// TIA Portal V17 export
// export: Created 2022-07-20T07:01:26.6168185Z, ExportSetting WithDefaults, DisplayName Totally Integrated Automation Portal, DisplayVersion V17, DisplayName TIA Portal Openness, DisplayVersion V17, DisplayName TIA Portal Version Control Interface, DisplayVersion V17, DisplayName SINAMICS Startdrive Advanced, DisplayVersion V17, DisplayName SINAMICS Startdrive G130, G150, S120, S150, SINAMICS MV, S210, DisplayVersion V17, DisplayName SINAMICS Startdrive G110M, G120, G120C, G120D, G120P, G115D, DisplayVersion V17, DisplayName STEP 7 Professional, DisplayVersion V17, DisplayName STEP 7 Safety, DisplayVersion V17, DisplayName WinCC Advanced, DisplayVersion V17
FUNCTION_BLOCK "FB10234_LexiumMotor"   // FB10234, LAD
{ S7_Optimized_Access := 'TRUE' }
VERSION : 0.1
// stored: AutoNumber false, IsIECCheckEnabled false, IsRetainMemResEnabled false, MemoryReserve 100, SetENOAutomatically false, UDAEnableTagReadback false
   VAR_INPUT
      Drive_In : "TLexium_MDrv_Drv2Plc";
      RequestAcknowledge : Bool;
      RequestHoming : Bool;
      ScaleInverted : Bool;
      RequestGoToAbsolutePosition_1 : Bool;
      RequestGoToAbsolutePosition_2 : Bool;
      RequestGoToAbsolutePosition_3 : Bool;
      RequestGoToAbsolutePosition_4 : Bool;
      RequestGoToAbsolutePosition_5 : Bool;
      RequestGoToAbsolutePosition_6 : Bool;
      RequestGoToAbsolutePosition_7 : Bool;
      RequestGoToAbsolutePosition_8 : Bool;
      RequestGoToAbsolutePosition_9 : Bool;
      RequestGoToAbsolutePosition_10 : Bool;
      RequestGoToRelativePosition : Bool;
      RequestJogBackward : Bool;
      RequestJogForward : Bool;
      RequestStop : Bool;
      AbsolutePosition_1 : Real;
      AbsolutePosition_2 : Real;
      AbsolutePosition_3 : Real;
      AbsolutePosition_4 : Real;
      AbsolutePosition_5 : Real;
      AbsolutePosition_6 : Real;
      AbsolutePosition_7 : Real;
      AbsolutePosition_8 : Real;
      AbsolutePosition_9 : Real;
      AbsolutePosition_10 : Real;
      HoldCurrent : SInt;
      RunCurrent : SInt;
      StepResolution : UInt := 25;
      StepsByMotorTurn : DInt := 200;
      MmByMotorTurn : LReal;
      "InitialVelocity_mm.s-1" : Real;
      "HomingVelocity_mm.s-1" : DInt;
      "Velocity_mm.s-1" : Real;
      "JogVelocity_mm.s-1" : Real;
      "Acceleration_mm.s-2" : Real;
      "Deceleration_mm.s-2" : Real;
   END_VAR
   VAR_OUTPUT
      ActualPosition_mm : Real;
      MotorInMovement : Bool;
      HomingInProgress : Bool;
      HomingDone : Bool;
      IsInAbsolutePosition_1 { ExternalAccessible := 'False'; ExternalVisible := 'False'; ExternalWritable := 'False'} : Bool;
      IsInAbsolutePosition_2 { ExternalAccessible := 'False'; ExternalVisible := 'False'; ExternalWritable := 'False'} : Bool;
      IsInAbsolutePosition_3 { ExternalAccessible := 'False'; ExternalVisible := 'False'; ExternalWritable := 'False'} : Bool;
      IsInAbsolutePosition_4 { ExternalAccessible := 'False'; ExternalVisible := 'False'; ExternalWritable := 'False'} : Bool;
      IsInAbsolutePosition_5 { ExternalAccessible := 'False'; ExternalVisible := 'False'; ExternalWritable := 'False'} : Bool;
      IsInAbsolutePosition_6 { ExternalAccessible := 'False'; ExternalVisible := 'False'; ExternalWritable := 'False'} : Bool;
      IsInAbsolutePosition_7 { ExternalAccessible := 'False'; ExternalVisible := 'False'; ExternalWritable := 'False'} : Bool;
      IsInAbsolutePosition_8 { ExternalAccessible := 'False'; ExternalVisible := 'False'; ExternalWritable := 'False'} : Bool;
      IsInAbsolutePosition_9 { ExternalAccessible := 'False'; ExternalVisible := 'False'; ExternalWritable := 'False'} : Bool;
      IsInAbsolutePosition_10 { ExternalAccessible := 'False'; ExternalVisible := 'False'; ExternalWritable := 'False'} : Bool;
      IsInAbsoluteMicrostepPosition_1 : Bool;
      IsInAbsoluteMicrostepPosition_2 : Bool;
      IsInAbsoluteMicrostepPosition_3 : Bool;
      IsInAbsoluteMicrostepPosition_4 : Bool;
      IsInAbsoluteMicrostepPosition_5 : Bool;
      IsInAbsoluteMicrostepPosition_6 : Bool;
      IsInAbsoluteMicrostepPosition_7 : Bool;
      IsInAbsoluteMicrostepPosition_8 : Bool;
      IsInAbsoluteMicrostepPosition_9 : Bool;
      IsInAbsoluteMicrostepPosition_10 : Bool;
      Busy : Bool;
      StatusCode : UInt;
      Error : Bool;
      ErrorCode : Array[0..9] of UInt;
   END_VAR
   VAR_IN_OUT
      Drive_Out : "TLexium_MDrv_Plc2Drv";
   END_VAR
   VAR
      SendJog : Bool;
      Static_InError : Bool;
      HomingErrorDetected : Bool;
      AcknowledgeHomingError : Bool;
      AcknowledgeStopError : Bool;
      SendHomingType : Bool;
      SendHomingPosition : Bool;
      SendAbsolutePosition : Bool;
      LockedRotorFaultDetected : Bool;
      i : USInt;
      NumberOfErrorDetected : USInt;
      MotorMovementStateDiagram : Int;
      Static_ErrorCode : UInt;
      MaxVelocity : DWord;
      AbsoluteMicrostepPosition_1 : LInt;
      AbsoluteMicrostepPosition_2 : LInt;
      AbsoluteMicrostepPosition_3 : LInt;
      AbsoluteMicrostepPosition_4 : LInt;
      AbsoluteMicrostepPosition_5 : LInt;
      AbsoluteMicrostepPosition_6 : LInt;
      AbsoluteMicrostepPosition_7 : LInt;
      AbsoluteMicrostepPosition_8 : LInt;
      AbsoluteMicrostepPosition_9 : LInt;
      AbsoluteMicrostepPosition_10 : LInt;
      R_TRIG_MotorAcknowledge : R_TRIG;
      R_TRIG_ChangeMicrostepResolution : R_TRIG;
      R_TRIG_ChangeInitialVelocity : R_TRIG;
      R_TRIG_ChangeVelocity : R_TRIG;
      R_TRIG_ChangeJogVelocity : R_TRIG;
      R_TRIG_ChangeAcceleration : R_TRIG;
      R_TRIG_ChangeDeceleration { S7_SetPoint := 'True'} : R_TRIG;
      R_TRIG_ChangeRunCurrent : R_TRIG;
      R_TRIG_ChangeHoldCurrent : R_TRIG;
      R_TRIG_RequestHoming { S7_SetPoint := 'True'} : R_TRIG;
      R_TRIG_RequestGoToPosition_1 { S7_SetPoint := 'True'} : R_TRIG;
      R_TRIG_RequestGoToPosition_2 { S7_SetPoint := 'True'} : R_TRIG;
      R_TRIG_RequestGoToPosition_3 { S7_SetPoint := 'True'} : R_TRIG;
      R_TRIG_RequestGoToPosition_4 { S7_SetPoint := 'True'} : R_TRIG;
      R_TRIG_RequestGoToPosition_5 { S7_SetPoint := 'True'} : R_TRIG;
      R_TRIG_RequestGoToPosition_6 { S7_SetPoint := 'True'} : R_TRIG;
      R_TRIG_RequestGoToPosition_7 { S7_SetPoint := 'True'} : R_TRIG;
      R_TRIG_RequestGoToPosition_8 { S7_SetPoint := 'True'} : R_TRIG;
      R_TRIG_RequestGoToPosition_9 { S7_SetPoint := 'True'} : R_TRIG;
      R_TRIG_RequestGoToPosition_10 { S7_SetPoint := 'True'} : R_TRIG;
      R_TRIG_RequestJogForward { S7_SetPoint := 'True'} : R_TRIG;
      R_TRIG_RequestJogBackward { S7_SetPoint := 'True'} : R_TRIG;
      R_TRIG_RequestStop { S7_SetPoint := 'True'} : R_TRIG;
      R_TRIG_MotorStopped { S7_SetPoint := 'True'} : R_TRIG;
      R_TRIG_MotorMovementDone { S7_SetPoint := 'True'} : R_TRIG;
      R_TRIG_ScaleInverted { S7_SetPoint := 'True'} : R_TRIG;
      R_TRIG_ErrorCodeChanged { S7_SetPoint := 'True'} : R_TRIG;
      R_TRIG_HomingErrorDetected { S7_SetPoint := 'True'} : R_TRIG;
      F_TRIG_RequestJogForward { S7_SetPoint := 'True'} : F_TRIG;
      F_TRIG_RequestJogBackward { S7_SetPoint := 'True'} : F_TRIG;
      TON_MotorHM { S7_SetPoint := 'True'} : TON_TIME;
      TON_MotorEnabled : TON_TIME;
      TON_MotorNotEnabled { S7_SetPoint := 'True'} : TOF_TIME;
      TON_MotorNotMoving { S7_SetPoint := 'True'} : TOF_TIME;
      TON_MotorHomingMovementDone { S7_SetPoint := 'True'} : TON_TIME;
      TON_MotorStopped { S7_SetPoint := 'True'} : TON_TIME;
      TON_IsInAbsolutePosition { S7_SetPoint := 'True'} : TON_TIME;
      TON_RetractSensorTimeout { S7_SetPoint := 'True'} : TON_TIME;
      FB10003_Pulse_SendHoldCurrent { S7_SetPoint := 'True'} : "FB10003_Pulse";
      FB10003_Pulse_SendRunCurrent { S7_SetPoint := 'True'} : "FB10003_Pulse";
      FB10003_Pulse_SendDeceleration { S7_SetPoint := 'True'} : "FB10003_Pulse";
      FB10003_Pulse_SendAcceleration { S7_SetPoint := 'True'} : "FB10003_Pulse";
      FB10003_Pulse_SendMicrostepResolution { S7_SetPoint := 'True'} : "FB10003_Pulse";
      FB10003_Pulse_SendInitialVelocity { S7_SetPoint := 'True'} : "FB10003_Pulse";
      FB10003_Pulse_SendVelocity { S7_SetPoint := 'True'} : "FB10003_Pulse";
      FB10003_Pulse_SendHoming { S7_SetPoint := 'True'} : "FB10003_Pulse";
      FB10003_Pulse_SendHomingPosition { S7_SetPoint := 'True'} : "FB10003_Pulse";
      FB10003_Pulse_SendAbsolutePosition { S7_SetPoint := 'True'} : "FB10003_Pulse";
      FB10003_Pulse_SendJog { S7_SetPoint := 'True'} : "FB10003_Pulse";
      FB10003_Pulse_SendMode { S7_SetPoint := 'True'} : "FB10003_Pulse";
      FB10003_Pulse_SendAcknowledge { S7_SetPoint := 'True'} : "FB10003_Pulse";
      FB10003_Pulse_SendScaleDirection { S7_SetPoint := 'True'} : "FB10003_Pulse";
   END_VAR
   VAR CONSTANT
      WAIT_FOR_MOTOR_MOVEMENT_REQUESTS : Int := 0;
      MOTOR_DISABLE : Int := 10;
      HOMING_TYPE : Int := 15;
      HOMING_MOVEMENT : Int := 20;
      HOMING_ACKNOWLEDGE_HOMING_ERROR : Int := 30;
      HOMING_WAIT_FOR_MOTOR_NOT_ENABLE : Int := 40;
      HOMING_SET_POSITION : Int := 50;
      GO_TO_ABSOLUTE_POSITION_1 : Int := 60;
      GO_TO_ABSOLUTE_POSITION_2 : Int := 70;
      GO_TO_ABSOLUTE_POSITION_3 : Int := 80;
      GO_TO_ABSOLUTE_POSITION_4 : Int := 90;
      GO_TO_ABSOLUTE_POSITION_5 : Int := 100;
      GO_TO_ABSOLUTE_POSITION_6 : Int := 110;
      GO_TO_ABSOLUTE_POSITION_7 : Int := 120;
      GO_TO_ABSOLUTE_POSITION_8 : Int := 130;
      GO_TO_ABSOLUTE_POSITION_9 : Int := 140;
      SET_ABSOLUTE_POSITION_10 : Int := 150;
      JOG_FORWARD : Int := 160;
      JOG_BACKWARD : Int := 170;
      STOP_JOG : Int := 180;
      STOP : Int := 190;
      MOTOR_MOVEMENT_DONE : Int := 200;
   END_VAR
BEGIN

REGION Network 1 (SCL): First Scan
   IF "FirstScan" THEN
       #HomingDone := FALSE;
       #HomingInProgress := FALSE;
       FOR #i := 0 TO 9 DO
           #ErrorCode[#i] := 0;
       END_FOR;
       #NumberOfErrorDetected := 0;
       #HomingErrorDetected := FALSE;
   END_IF;
END_REGION

REGION Network 2 (SCL): Edge Signals & Timers
   REGION EDGE SIGNALS
       #R_TRIG_ChangeInitialVelocity(CLK := #Drive_In.VI <> #Drive_Out.VI);
       #R_TRIG_ChangeVelocity(CLK := #Drive_In.VM <> #Drive_Out.VM);
       //#R_TRIG_ChangeJogVelocity(CLK := #Drive_In.SL <> #Drive_Out.SL);
       #R_TRIG_ChangeAcceleration(CLK := #Drive_In.A <> #Drive_Out.A);
       #R_TRIG_ChangeDeceleration(CLK := #Drive_In.D <> #Drive_Out.D);
       #R_TRIG_ChangeHoldCurrent(CLK := #Drive_In.HC <> #Drive_Out.HC);
       #R_TRIG_ChangeRunCurrent(CLK := #Drive_In.RC <> #Drive_Out.RC);
       #R_TRIG_RequestHoming(CLK := #RequestHoming AND #MotorMovementStateDiagram = #WAIT_FOR_MOTOR_MOVEMENT_REQUESTS);
       #R_TRIG_RequestGoToPosition_1(CLK := #RequestGoToAbsolutePosition_1 AND #MotorMovementStateDiagram = #WAIT_FOR_MOTOR_MOVEMENT_REQUESTS AND NOT(#IsInAbsoluteMicrostepPosition_1));
       #R_TRIG_RequestGoToPosition_2(CLK := #RequestGoToAbsolutePosition_2 AND #MotorMovementStateDiagram = #WAIT_FOR_MOTOR_MOVEMENT_REQUESTS AND NOT(#IsInAbsoluteMicrostepPosition_2));
       #R_TRIG_RequestGoToPosition_3(CLK := #RequestGoToAbsolutePosition_3 AND #MotorMovementStateDiagram = #WAIT_FOR_MOTOR_MOVEMENT_REQUESTS AND NOT(#IsInAbsoluteMicrostepPosition_3));
       #R_TRIG_RequestGoToPosition_4(CLK := #RequestGoToAbsolutePosition_4 AND #MotorMovementStateDiagram = #WAIT_FOR_MOTOR_MOVEMENT_REQUESTS AND NOT(#IsInAbsoluteMicrostepPosition_4));
       #R_TRIG_RequestGoToPosition_5(CLK := #RequestGoToAbsolutePosition_5 AND #MotorMovementStateDiagram = #WAIT_FOR_MOTOR_MOVEMENT_REQUESTS AND NOT(#IsInAbsoluteMicrostepPosition_5));
       #R_TRIG_RequestGoToPosition_6(CLK := #RequestGoToAbsolutePosition_6 AND #MotorMovementStateDiagram = #WAIT_FOR_MOTOR_MOVEMENT_REQUESTS AND NOT(#IsInAbsoluteMicrostepPosition_6));
       #R_TRIG_RequestGoToPosition_7(CLK := #RequestGoToAbsolutePosition_7 AND #MotorMovementStateDiagram = #WAIT_FOR_MOTOR_MOVEMENT_REQUESTS AND NOT(#IsInAbsoluteMicrostepPosition_7));
       #R_TRIG_RequestGoToPosition_8(CLK := #RequestGoToAbsolutePosition_8 AND #MotorMovementStateDiagram = #WAIT_FOR_MOTOR_MOVEMENT_REQUESTS AND NOT(#IsInAbsoluteMicrostepPosition_8));
       #R_TRIG_RequestGoToPosition_9(CLK := #RequestGoToAbsolutePosition_9 AND #MotorMovementStateDiagram = #WAIT_FOR_MOTOR_MOVEMENT_REQUESTS AND NOT(#IsInAbsoluteMicrostepPosition_9));
       #R_TRIG_RequestGoToPosition_10(CLK := #RequestGoToAbsolutePosition_10 AND #MotorMovementStateDiagram = #WAIT_FOR_MOTOR_MOVEMENT_REQUESTS AND NOT(#IsInAbsoluteMicrostepPosition_10));
       #R_TRIG_RequestJogBackward(CLK := #RequestJogBackward AND #MotorMovementStateDiagram = #WAIT_FOR_MOTOR_MOVEMENT_REQUESTS);
       #R_TRIG_RequestJogForward(CLK := #RequestJogForward AND #MotorMovementStateDiagram = #WAIT_FOR_MOTOR_MOVEMENT_REQUESTS);
       #R_TRIG_MotorStopped(CLK := #Drive_In.MV = 0);
       #R_TRIG_RequestStop(CLK := #RequestStop OR (#Drive_In.DE = 1 AND #Drive_In.ER <> 0 AND NOT(#Drive_In.ER = 85 AND #HomingInProgress)));
       #R_TRIG_MotorMovementDone(CLK := #TON_MotorNotEnabled.Q);
       #R_TRIG_ScaleInverted(CLK := #Drive_In.RD <> BOOL_TO_UINT(#ScaleInverted));
       #R_TRIG_ErrorCodeChanged(CLK := #Drive_In.ER <> #Static_ErrorCode);
       #R_TRIG_HomingErrorDetected(CLK := #HomingErrorDetected);

       #F_TRIG_RequestJogBackward(CLK := #RequestJogBackward);
       #F_TRIG_RequestJogForward(CLK := #RequestJogForward);
   END_REGION

   REGION TIMERS
       #TON_MotorEnabled(IN := #Drive_In.DE = 1,
                         PT := T#200ms);
       #TON_MotorHomingMovementDone(IN := #Drive_In.MV = 0 AND #MotorMovementStateDiagram = #HOMING_MOVEMENT,
                                    PT := T#1s);
       #TON_MotorStopped(IN := #MotorMovementStateDiagram = #STOP,
                         PT := T#1s);
       #TON_MotorNotMoving(IN := #Drive_In.MV = 0,
                           PT := T#200ms);
       #TON_MotorNotEnabled(IN := #Drive_In.DE = 0,
                            PT := T#200ms);
       #TON_RetractSensorTimeout(IN := #MotorMovementStateDiagram = #HOMING_MOVEMENT,
                                 PT := T#1000s);

       #TON_MotorHM(IN := #MotorMovementStateDiagram = #HOMING_TYPE,
                    PT := T#200ms);
   END_REGION
END_REGION

REGION Network 3 (SCL): Motor Commands Management
   #AbsoluteMicrostepPosition_1 := (TRUNC_LINT(#AbsolutePosition_1 * 10) * (#StepResolution * #StepsByMotorTurn) * 100) / (TRUNC_LINT(#MmByMotorTurn * 100) * 10);
   #AbsoluteMicrostepPosition_2 := (TRUNC_LINT(#AbsolutePosition_2 * 10) * (#StepResolution * #StepsByMotorTurn) * 100) / (TRUNC_LINT(#MmByMotorTurn * 100) * 10);
   #AbsoluteMicrostepPosition_3 := (TRUNC_LINT(#AbsolutePosition_3 * 10) * (#StepResolution * #StepsByMotorTurn) * 100) / (TRUNC_LINT(#MmByMotorTurn * 100) * 10);
   #AbsoluteMicrostepPosition_4 := (TRUNC_LINT(#AbsolutePosition_4 * 10) * (#StepResolution * #StepsByMotorTurn) * 100) / (TRUNC_LINT(#MmByMotorTurn * 100) * 10);
   #AbsoluteMicrostepPosition_5 := (TRUNC_LINT(#AbsolutePosition_5 * 10) * (#StepResolution * #StepsByMotorTurn) * 100) / (TRUNC_LINT(#MmByMotorTurn * 100) * 10);
   #AbsoluteMicrostepPosition_6 := (TRUNC_LINT(#AbsolutePosition_6 * 10) * (#StepResolution * #StepsByMotorTurn) * 100) / (TRUNC_LINT(#MmByMotorTurn * 100) * 10);
   #AbsoluteMicrostepPosition_7 := (TRUNC_LINT(#AbsolutePosition_7 * 10) * (#StepResolution * #StepsByMotorTurn) * 100) / (TRUNC_LINT(#MmByMotorTurn * 100) * 10);
   #AbsoluteMicrostepPosition_8 := (TRUNC_LINT(#AbsolutePosition_8 * 10) * (#StepResolution * #StepsByMotorTurn) * 100) / (TRUNC_LINT(#MmByMotorTurn * 100) * 10);
   #AbsoluteMicrostepPosition_9 := (TRUNC_LINT(#AbsolutePosition_9 * 10) * (#StepResolution * #StepsByMotorTurn) * 100) / (TRUNC_LINT(#MmByMotorTurn * 100) * 10);
   #AbsoluteMicrostepPosition_10 := (TRUNC_LINT(#AbsolutePosition_10 * 10) * (#StepResolution * #StepsByMotorTurn) * 100) / (TRUNC_LINT(#MmByMotorTurn * 100) * 10);
END_REGION

REGION Network 4 (SCL): Motor Error Management
   //Acknowledge Management
   IF #Drive_In.ER = 104 THEN
       #LockedRotorFaultDetected := TRUE;
   ELSIF #Drive_In.ER = 0 THEN
       #LockedRotorFaultDetected := FALSE;
   END_IF;
   #Drive_Out.CF := BOOL_TO_SINT((#RequestAcknowledge OR #AcknowledgeHomingError OR #RequestStop) AND #LockedRotorFaultDetected);
   IF #RequestAcknowledge OR #AcknowledgeHomingError OR #AcknowledgeStopError THEN
       FOR #i := 0 TO 9 DO
           #ErrorCode[#i] := 0;
       END_FOR;
       #Drive_Out.ER := 0;
       #Error := FALSE;
       #NumberOfErrorDetected := 0;
       #HomingErrorDetected := FALSE;
   END_IF;
END_REGION

REGION Network 5 (SCL): Motor Communucation Management
   REGION MODE
       #Drive_Out.AS := 2;
       #FB10003_Pulse_SendMode(CLK := "FirstScan",
                               PT := T#50ms,
                               Q := #Drive_Out.Toggle_reg_17);
   END_REGION

   REGION MICROSTEP RESOLUTION
       #Drive_Out.MS := #StepResolution;
       #FB10003_Pulse_SendMicrostepResolution(CLK := "FirstScan",
                                              PT := T#50ms,
                                              Q := #Drive_Out.Toggle_reg_14);
   END_REGION

   REGION INITIAL VELOCITY
       #Drive_Out.VI := DINT_TO_DWORD(REAL_TO_DINT(#"InitialVelocity_mm.s-1" * UINT_TO_REAL(#StepResolution) * DINT_TO_REAL(#StepsByMotorTurn) * 100.0) / TRUNC(#MmByMotorTurn * 100));
       #FB10003_Pulse_SendInitialVelocity(CLK := "FirstScan" OR #R_TRIG_ChangeInitialVelocity.Q,
                                          PT := T#50ms,
                                          Q := #Drive_Out.Toggle_reg_4);
   END_REGION

   REGION VELOCITY
       #Drive_Out.VM := DINT_TO_DWORD(REAL_TO_DINT(#"Velocity_mm.s-1" * UINT_TO_REAL(#StepResolution) * DINT_TO_REAL(#StepsByMotorTurn) * 100.0) / TRUNC(#MmByMotorTurn * 100));
       IF #Drive_Out.VM > DINT_TO_DWORD(UINT_TO_DINT(#StepResolution) * 10000) THEN
           #Drive_Out.VM := (#StepResolution * 10000) - 1;
       ELSIF #Drive_Out.VM < #Drive_Out.VI THEN
           #Drive_Out.VM := #Drive_Out.VI + 1;
       END_IF;
       #FB10003_Pulse_SendVelocity(CLK := "FirstScan" OR #R_TRIG_ChangeVelocity.Q,
                                   PT := T#50ms,
                                   Q := #Drive_Out.Toggle_reg_5);
   END_REGION

   REGION ACCELERATION
       #Drive_Out.A := DINT_TO_DWORD(REAL_TO_DINT(#"Acceleration_mm.s-2" * UINT_TO_REAL(#StepResolution) * DINT_TO_REAL(#StepsByMotorTurn) * 100.0) / TRUNC(#MmByMotorTurn * 100));
       #FB10003_Pulse_SendAcceleration(CLK := "FirstScan" OR #R_TRIG_ChangeAcceleration.Q,
                                       PT := T#50ms,
                                       Q := #Drive_Out.Toggle_reg_1);
   END_REGION

   REGION DECELERATION
       #Drive_Out.D := DINT_TO_DWORD(REAL_TO_DINT(#"Deceleration_mm.s-2" * UINT_TO_REAL(#StepResolution) * DINT_TO_REAL(#StepsByMotorTurn) * 100.0) / TRUNC(#MmByMotorTurn * 100));
       #FB10003_Pulse_SendDeceleration(CLK := "FirstScan" OR #R_TRIG_ChangeDeceleration.Q,
                                       PT := T#50ms,
                                       Q := #Drive_Out.Toggle_reg_2);
   END_REGION

   REGION HOLD CURRENT
       IF #HoldCurrent > 100 THEN
           #Drive_Out.HC := 100;
       ELSIF #HoldCurrent < 0 THEN
           #Drive_Out.HC := 0;
       ELSE
           #Drive_Out.HC := #HoldCurrent;
       END_IF;
       #FB10003_Pulse_SendHoldCurrent(CLK := "FirstScan" OR #R_TRIG_ChangeHoldCurrent.Q,
                                      PT := T#50ms,
                                      Q := #Drive_Out.Toggle_reg_18);
   END_REGION

   REGION RUN CURRENT
       IF #RunCurrent > 100 THEN
           #Drive_Out.RC := 100;
       ELSIF #RunCurrent < 0 THEN
           #Drive_Out.RC := 0;
       ELSE
           #Drive_Out.RC := #RunCurrent;
       END_IF;
       #FB10003_Pulse_SendRunCurrent(CLK := "FirstScan" OR #R_TRIG_ChangeRunCurrent.Q,
                                     PT := T#50ms,
                                     Q := #Drive_Out.Toggle_reg_20);
   END_REGION

   REGION HOMING TYPE   
       #FB10003_Pulse_SendHoming(CLK := #TON_MotorEnabled.Q AND #SendHomingType,
                                 PT := T#50ms,
                                 Q := #Drive_Out.Toggle_reg_22);
   END_REGION

   REGION HOMING POSITION
       #FB10003_Pulse_SendHomingPosition(CLK := #TON_MotorNotEnabled.Q AND #SendHomingPosition,
                                         PT := T#50ms,
                                         Q := #Drive_Out.Toggle_reg_12);
   END_REGION

   REGION ABSOLUTE POSITION
       #FB10003_Pulse_SendAbsolutePosition(CLK := #TON_MotorEnabled.Q AND #SendAbsolutePosition,
                                           PT := T#50ms,
                                           Q := #Drive_Out.Toggle_reg_9);
   END_REGION

   REGION JOG
       #FB10003_Pulse_SendJog(CLK := #SendJog,
                              PT := T#50ms,
                              Q := #Drive_Out.Toggle_reg_11);
   END_REGION

   REGION ACKNOWLEDGE
       #FB10003_Pulse_SendAcknowledge(CLK := (#RequestAcknowledge AND NOT (#Error)) OR
                                      (#AcknowledgeHomingError AND NOT (#Error)) OR
                                      #RequestStop OR
                                      "FirstScan",
                                      PT := T#50ms,
                                      Q := #Drive_Out.Toggle_reg_15);
   END_REGION

   REGION SCALE DIRECTION
       IF #R_TRIG_ScaleInverted.Q THEN
           #Drive_Out.RD := BOOL_TO_UINT(#ScaleInverted);
       END_IF;
       #FB10003_Pulse_SendScaleDirection(CLK := (#Drive_Out.RD <> #Drive_In.RD) AND #Drive_In.DE = 0,
                                         PT := T#50ms,
                                         Q := #Drive_Out.Toggle_reg_16);
   END_REGION
END_REGION

REGION Network 6 (SCL): Motor Movement Management
   IF #R_TRIG_RequestStop.Q AND #Drive_In.DE = 1 THEN
       #MotorMovementStateDiagram := #STOP;
   END_IF;

   CASE #MotorMovementStateDiagram OF
       #WAIT_FOR_MOTOR_MOVEMENT_REQUESTS:
           IF #R_TRIG_RequestHoming.Q THEN
               #HomingDone := FALSE;
               #Drive_Out.DE := 1;
               #MotorMovementStateDiagram := #HOMING_TYPE;
           ELSIF #R_TRIG_RequestGoToPosition_1.Q THEN
               #Drive_Out.DE := 1;
               #MotorMovementStateDiagram := #GO_TO_ABSOLUTE_POSITION_1;
           ELSIF #R_TRIG_RequestGoToPosition_2.Q THEN
               #Drive_Out.DE := 1;
               #MotorMovementStateDiagram := #GO_TO_ABSOLUTE_POSITION_2;
           ELSIF #R_TRIG_RequestGoToPosition_3.Q THEN
               #Drive_Out.DE := 1;
               #MotorMovementStateDiagram := #GO_TO_ABSOLUTE_POSITION_3;
           ELSIF #R_TRIG_RequestGoToPosition_4.Q THEN
               #Drive_Out.DE := 1;
               #MotorMovementStateDiagram := #GO_TO_ABSOLUTE_POSITION_4;
           ELSIF #R_TRIG_RequestGoToPosition_5.Q THEN
               #Drive_Out.DE := 1;
               #MotorMovementStateDiagram := #GO_TO_ABSOLUTE_POSITION_5;
           ELSIF #R_TRIG_RequestGoToPosition_6.Q THEN
               #Drive_Out.DE := 1;
               #MotorMovementStateDiagram := #GO_TO_ABSOLUTE_POSITION_6;
           ELSIF #R_TRIG_RequestGoToPosition_7.Q THEN
               #Drive_Out.DE := 1;
               #MotorMovementStateDiagram := #GO_TO_ABSOLUTE_POSITION_7;
           ELSIF #R_TRIG_RequestGoToPosition_8.Q THEN
               #Drive_Out.DE := 1;
               #MotorMovementStateDiagram := #GO_TO_ABSOLUTE_POSITION_8;
           ELSIF #R_TRIG_RequestGoToPosition_9.Q THEN
               #Drive_Out.DE := 1;
               #MotorMovementStateDiagram := #GO_TO_ABSOLUTE_POSITION_9;
           ELSIF #R_TRIG_RequestGoToPosition_10.Q THEN
               #Drive_Out.DE := 1;
               #MotorMovementStateDiagram := #SET_ABSOLUTE_POSITION_10;
           ELSIF #R_TRIG_RequestJogBackward.Q THEN
               #Drive_Out.DE := 1;
               #MotorMovementStateDiagram := #JOG_BACKWARD;
           ELSIF #R_TRIG_RequestJogForward.Q THEN
               #Drive_Out.DE := 1;
               #MotorMovementStateDiagram := #JOG_FORWARD;
           END_IF;
       #HOMING_TYPE:
           IF #TON_MotorEnabled.Q THEN
               #Drive_Out.HM := 1;

               IF #TON_MotorHM.Q THEN
                   RESET_TIMER(#TON_MotorHM);
                   #MotorMovementStateDiagram := #HOMING_MOVEMENT;
               END_IF;
           END_IF;
       #HOMING_MOVEMENT:
           IF #TON_MotorEnabled.Q THEN
               #MotorInMovement := TRUE;
               #HomingInProgress := TRUE;
               #SendHomingType := TRUE;
               IF #TON_MotorHomingMovementDone.Q THEN
                   #SendHomingType := FALSE;
                   #MotorMovementStateDiagram := #HOMING_WAIT_FOR_MOTOR_NOT_ENABLE;
               ELSIF #TON_RetractSensorTimeout.Q THEN
                   #SendHomingType := FALSE;
                   #HomingErrorDetected := TRUE;
                   #MotorMovementStateDiagram := #STOP;
               END_IF;
           END_IF;
       #HOMING_WAIT_FOR_MOTOR_NOT_ENABLE:
           #Drive_Out.DE := 0;

           //Condition To Go To Next Step
           IF #TON_MotorNotEnabled.Q THEN
               #MotorMovementStateDiagram := #HOMING_ACKNOWLEDGE_HOMING_ERROR;
           END_IF;
       #HOMING_ACKNOWLEDGE_HOMING_ERROR:
           IF #Drive_In.ER <> 0 THEN //IF #Drive_In.ER = 85 THEN
               #AcknowledgeHomingError := "Clock_0.5Hz";
           END_IF;
           IF #Drive_In.ER = 0 THEN
               #AcknowledgeHomingError := FALSE;
               #MotorMovementStateDiagram := #HOMING_SET_POSITION;
           END_IF;
       #HOMING_SET_POSITION:
           IF #TON_MotorNotEnabled.Q THEN
               #Drive_Out.P := 0;
               #SendHomingPosition := NOT(#Drive_In.P = 0) AND "Clock_0.5Hz";
               IF #Drive_In.P = 0 THEN
                   #MotorInMovement := FALSE;
                   #HomingInProgress := FALSE;
                   #SendHomingPosition := FALSE;
                   #HomingDone := TRUE;
                   #MotorMovementStateDiagram := #MOTOR_MOVEMENT_DONE;
               END_IF;
           END_IF;
       #GO_TO_ABSOLUTE_POSITION_1:
           IF #TON_MotorEnabled.Q THEN
               #MotorInMovement := TRUE;
               #Drive_Out.MA := LINT_TO_DINT(#AbsoluteMicrostepPosition_1);
               #SendAbsolutePosition := NOT (SINT_TO_BOOL(#Drive_In.MV)) AND NOT (#IsInAbsoluteMicrostepPosition_1) AND "Clock_0.5Hz";;
               IF #IsInAbsoluteMicrostepPosition_1 THEN
                   #MotorInMovement := FALSE;
                   #SendAbsolutePosition := FALSE;
                   #Drive_Out.DE := 0;
               END_IF;
           ELSIF #R_TRIG_MotorMovementDone.Q THEN
               #MotorMovementStateDiagram := #MOTOR_MOVEMENT_DONE;
           END_IF;
       #GO_TO_ABSOLUTE_POSITION_2:
           IF #TON_MotorEnabled.Q THEN
               #MotorInMovement := TRUE;
               #Drive_Out.MA := LINT_TO_DINT(#AbsoluteMicrostepPosition_2);
               #SendAbsolutePosition := NOT (SINT_TO_BOOL(#Drive_In.MV)) AND NOT (#IsInAbsoluteMicrostepPosition_2) AND "Clock_0.5Hz";;
               IF #IsInAbsoluteMicrostepPosition_2 THEN
                   #MotorInMovement := FALSE;
                   #SendAbsolutePosition := FALSE;
                   #Drive_Out.DE := 0;
               END_IF;
           ELSIF #R_TRIG_MotorMovementDone.Q THEN
               #MotorMovementStateDiagram := #MOTOR_MOVEMENT_DONE;
           END_IF;
       #GO_TO_ABSOLUTE_POSITION_3:
           IF #TON_MotorEnabled.Q THEN
               #MotorInMovement := TRUE;
               #Drive_Out.MA := LINT_TO_DINT(#AbsoluteMicrostepPosition_3);
               #SendAbsolutePosition := NOT (SINT_TO_BOOL(#Drive_In.MV)) AND NOT (#IsInAbsoluteMicrostepPosition_3) AND "Clock_0.5Hz";;
               IF #IsInAbsoluteMicrostepPosition_3 THEN
                   #MotorInMovement := FALSE;
                   #SendAbsolutePosition := FALSE;
                   #Drive_Out.DE := 0;
               END_IF;
           ELSIF #R_TRIG_MotorMovementDone.Q THEN
               #MotorMovementStateDiagram := #MOTOR_MOVEMENT_DONE;
           END_IF;
       #GO_TO_ABSOLUTE_POSITION_4:
           IF #TON_MotorEnabled.Q THEN
               #MotorInMovement := TRUE;
               #Drive_Out.MA := LINT_TO_DINT(#AbsoluteMicrostepPosition_4);
               #SendAbsolutePosition := NOT (SINT_TO_BOOL(#Drive_In.MV)) AND NOT (#IsInAbsoluteMicrostepPosition_4) AND "Clock_0.5Hz";;
               IF #IsInAbsoluteMicrostepPosition_4 THEN
                   #SendAbsolutePosition := FALSE;
                   #Drive_Out.DE := 0;
               END_IF;
           ELSIF #R_TRIG_MotorMovementDone.Q THEN
               #MotorMovementStateDiagram := #MOTOR_MOVEMENT_DONE;
           END_IF;
       #GO_TO_ABSOLUTE_POSITION_5:
           IF #TON_MotorEnabled.Q THEN
               #MotorInMovement := TRUE;
               #Drive_Out.MA := LINT_TO_DINT(#AbsoluteMicrostepPosition_5);
               #SendAbsolutePosition := NOT (SINT_TO_BOOL(#Drive_In.MV)) AND NOT (#IsInAbsoluteMicrostepPosition_5) AND "Clock_0.5Hz";;
               IF #IsInAbsoluteMicrostepPosition_5 THEN
                   #SendAbsolutePosition := FALSE;
                   #Drive_Out.DE := 0;
               END_IF;
           ELSIF #R_TRIG_MotorMovementDone.Q THEN
               #MotorMovementStateDiagram := #MOTOR_MOVEMENT_DONE;
           END_IF;
       #GO_TO_ABSOLUTE_POSITION_6:
           IF #TON_MotorEnabled.Q THEN
               #MotorInMovement := TRUE;
               #Drive_Out.MA := LINT_TO_DINT(#AbsoluteMicrostepPosition_6);
               #SendAbsolutePosition := NOT (SINT_TO_BOOL(#Drive_In.MV)) AND NOT (#IsInAbsoluteMicrostepPosition_6) AND "Clock_0.5Hz";;
               IF #IsInAbsoluteMicrostepPosition_6 THEN
                   #SendAbsolutePosition := FALSE;
                   #Drive_Out.DE := 0;
               END_IF;
           ELSIF #R_TRIG_MotorMovementDone.Q THEN
               #MotorMovementStateDiagram := #MOTOR_MOVEMENT_DONE;
           END_IF;
       #GO_TO_ABSOLUTE_POSITION_7:
           IF #TON_MotorEnabled.Q THEN
               #MotorInMovement := TRUE;
               #Drive_Out.MA := LINT_TO_DINT(#AbsoluteMicrostepPosition_7);
               #SendAbsolutePosition := NOT (SINT_TO_BOOL(#Drive_In.MV)) AND NOT (#IsInAbsoluteMicrostepPosition_7) AND "Clock_0.5Hz";;
               IF #IsInAbsoluteMicrostepPosition_7 THEN
                   #SendAbsolutePosition := FALSE;
                   #Drive_Out.DE := 0;
               END_IF;
           ELSIF #R_TRIG_MotorMovementDone.Q THEN
               #MotorMovementStateDiagram := #MOTOR_MOVEMENT_DONE;
           END_IF;
       #GO_TO_ABSOLUTE_POSITION_8:
           IF #TON_MotorEnabled.Q THEN
               #MotorInMovement := TRUE;
               #Drive_Out.MA := LINT_TO_DINT(#AbsoluteMicrostepPosition_8);
               #SendAbsolutePosition := NOT (SINT_TO_BOOL(#Drive_In.MV)) AND NOT (#IsInAbsoluteMicrostepPosition_8) AND "Clock_0.5Hz";;
               IF #IsInAbsoluteMicrostepPosition_8 THEN
                   #SendAbsolutePosition := FALSE;
                   #Drive_Out.DE := 0;
               END_IF;
           ELSIF #R_TRIG_MotorMovementDone.Q THEN
               #MotorMovementStateDiagram := #MOTOR_MOVEMENT_DONE;
           END_IF;
       #GO_TO_ABSOLUTE_POSITION_9:
           IF #TON_MotorEnabled.Q THEN
               #MotorInMovement := TRUE;
               #Drive_Out.MA := LINT_TO_DINT(#AbsoluteMicrostepPosition_9);
               #SendAbsolutePosition := NOT (SINT_TO_BOOL(#Drive_In.MV)) AND NOT (#IsInAbsoluteMicrostepPosition_9) AND "Clock_0.5Hz";;
               IF #IsInAbsoluteMicrostepPosition_9 THEN
                   #SendAbsolutePosition := FALSE;
                   #Drive_Out.DE := 0;
               END_IF;
           ELSIF #R_TRIG_MotorMovementDone.Q THEN
               #MotorMovementStateDiagram := #MOTOR_MOVEMENT_DONE;
           END_IF;
       #SET_ABSOLUTE_POSITION_10:
           IF #TON_MotorEnabled.Q THEN
               #MotorInMovement := TRUE;
               #Drive_Out.MA := LINT_TO_DINT(#AbsoluteMicrostepPosition_10);
               #SendAbsolutePosition := NOT (SINT_TO_BOOL(#Drive_In.MV)) AND NOT (#IsInAbsoluteMicrostepPosition_10) AND "Clock_0.5Hz";;
               IF #IsInAbsoluteMicrostepPosition_10 THEN
                   #SendAbsolutePosition := FALSE;
                   #Drive_Out.DE := 0;
               END_IF;
           ELSIF #R_TRIG_MotorMovementDone.Q THEN
               #MotorMovementStateDiagram := #MOTOR_MOVEMENT_DONE;
           END_IF;
       #JOG_BACKWARD:
           IF #TON_MotorEnabled.Q THEN
               #MotorInMovement := TRUE;
               #Drive_Out.SL := - REAL_TO_DINT(#"Velocity_mm.s-1" * UINT_TO_REAL(#StepResolution) * DINT_TO_REAL(#StepsByMotorTurn) * 100.0) / TRUNC(#MmByMotorTurn * 100);
               #SendJog := TRUE;
               IF #F_TRIG_RequestJogBackward.Q THEN
                   #SendJog := FALSE;
                   #MotorMovementStateDiagram := #STOP_JOG;
               END_IF;
           END_IF;
       #JOG_FORWARD:
           IF #TON_MotorEnabled.Q THEN
               #MotorInMovement := TRUE;
               #Drive_Out.SL := REAL_TO_DINT(#"Velocity_mm.s-1" * UINT_TO_REAL(#StepResolution) * DINT_TO_REAL(#StepsByMotorTurn) * 100.0) / TRUNC(#MmByMotorTurn * 100);
               #SendJog := TRUE;
               IF #F_TRIG_RequestJogForward.Q THEN
                   #SendJog := FALSE;
                   #MotorMovementStateDiagram := #STOP_JOG;
               END_IF;
           END_IF;
       #STOP_JOG:
           IF #TON_MotorEnabled.Q THEN
               #Drive_Out.SL := 0;
               #SendJog := TRUE;
               IF #TON_MotorNotMoving.Q THEN
                   #MotorInMovement := FALSE;
                   #SendJog := FALSE;
                   #Drive_Out.DE := 0;
               END_IF;
           ELSIF #R_TRIG_MotorMovementDone.Q THEN
               #MotorMovementStateDiagram := #MOTOR_MOVEMENT_DONE;
           END_IF;
       #STOP:
           IF #Drive_In.DE = 1 AND NOT(#Error) THEN
               #SendJog := TRUE;
           END_IF;
           #Drive_Out.SL := 0;
           #Drive_Out.DE := 0;
           #SendHomingPosition := FALSE;
           #SendAbsolutePosition := FALSE;
           //#Drive_Out.HM := 0;
           IF #TON_MotorNotEnabled.Q OR #TON_MotorStopped.Q THEN
               #HomingInProgress := FALSE;
               #MotorInMovement := FALSE;
               #SendJog := FALSE;
               #MotorMovementStateDiagram := #MOTOR_MOVEMENT_DONE;
           END_IF;
       #MOTOR_MOVEMENT_DONE:
           #MotorMovementStateDiagram := #WAIT_FOR_MOTOR_MOVEMENT_REQUESTS;
   END_CASE;
END_REGION

REGION Network 7 (SCL): Motor States Management
   #MotorInMovement := #Drive_In.MV = 1;

   #Busy := #MotorMovementStateDiagram > #WAIT_FOR_MOTOR_MOVEMENT_REQUESTS AND #MotorMovementStateDiagram < #MOTOR_MOVEMENT_DONE;

   IF #Drive_In.ER <> 0 AND NOT(#Drive_In.ER = 85 AND #HomingInProgress) THEN
       #Error := TRUE;
       #HomingDone := FALSE;
   END_IF;

   IF #R_TRIG_ErrorCodeChanged.Q THEN
       IF #NumberOfErrorDetected >= 0 AND #NumberOfErrorDetected <= 9 THEN
           #ErrorCode[#NumberOfErrorDetected] := #Drive_In.ER;
           #NumberOfErrorDetected += 1;
           #Static_ErrorCode := #Drive_In.ER;
       END_IF;

       IF #R_TRIG_HomingErrorDetected.Q THEN
           #ErrorCode[#NumberOfErrorDetected] := 200;
           #NumberOfErrorDetected += 1;
       END_IF;
   END_IF;

   #IsInAbsoluteMicrostepPosition_1 := "FC10021_TolerenceRelation"(X := #Drive_In.P, Y := #AbsoluteMicrostepPosition_1, Tolerance := LREAL_TO_REAL((DINT_TO_LREAL(#StepsByMotorTurn) * UINT_TO_LREAL(#StepResolution))/(#MmByMotorTurn*10)));
   #IsInAbsoluteMicrostepPosition_2 := "FC10021_TolerenceRelation"(X := #Drive_In.P, Y := #AbsoluteMicrostepPosition_2, Tolerance := LREAL_TO_REAL((DINT_TO_LREAL(#StepsByMotorTurn) * UINT_TO_LREAL(#StepResolution))/(#MmByMotorTurn*10)));
   #IsInAbsoluteMicrostepPosition_3 := "FC10021_TolerenceRelation"(X := #Drive_In.P, Y := #AbsoluteMicrostepPosition_3, Tolerance := LREAL_TO_REAL((DINT_TO_LREAL(#StepsByMotorTurn) * UINT_TO_LREAL(#StepResolution))/(#MmByMotorTurn*10)));
   #IsInAbsoluteMicrostepPosition_4 := "FC10021_TolerenceRelation"(X := #Drive_In.P, Y := #AbsoluteMicrostepPosition_4, Tolerance := LREAL_TO_REAL((DINT_TO_LREAL(#StepsByMotorTurn) * UINT_TO_LREAL(#StepResolution))/(#MmByMotorTurn*10)));
   #IsInAbsoluteMicrostepPosition_5 := "FC10021_TolerenceRelation"(X := #Drive_In.P, Y := #AbsoluteMicrostepPosition_5, Tolerance := LREAL_TO_REAL((DINT_TO_LREAL(#StepsByMotorTurn) * UINT_TO_LREAL(#StepResolution))/(#MmByMotorTurn*10)));
   #IsInAbsoluteMicrostepPosition_6 := "FC10021_TolerenceRelation"(X := #Drive_In.P, Y := #AbsoluteMicrostepPosition_6, Tolerance := LREAL_TO_REAL((DINT_TO_LREAL(#StepsByMotorTurn) * UINT_TO_LREAL(#StepResolution))/(#MmByMotorTurn*10)));
   #IsInAbsoluteMicrostepPosition_7 := "FC10021_TolerenceRelation"(X := #Drive_In.P, Y := #AbsoluteMicrostepPosition_7, Tolerance := LREAL_TO_REAL((DINT_TO_LREAL(#StepsByMotorTurn) * UINT_TO_LREAL(#StepResolution))/(#MmByMotorTurn*10)));
   #IsInAbsoluteMicrostepPosition_8 := "FC10021_TolerenceRelation"(X := #Drive_In.P, Y := #AbsoluteMicrostepPosition_8, Tolerance := LREAL_TO_REAL((DINT_TO_LREAL(#StepsByMotorTurn) * UINT_TO_LREAL(#StepResolution))/(#MmByMotorTurn*10)));
   #IsInAbsoluteMicrostepPosition_9 := "FC10021_TolerenceRelation"(X := #Drive_In.P, Y := #AbsoluteMicrostepPosition_9, Tolerance := LREAL_TO_REAL((DINT_TO_LREAL(#StepsByMotorTurn) * UINT_TO_LREAL(#StepResolution))/(#MmByMotorTurn*10)));
   #IsInAbsoluteMicrostepPosition_10 := "FC10021_TolerenceRelation"(X := #Drive_In.P, Y := #AbsoluteMicrostepPosition_10, Tolerance := LREAL_TO_REAL((DINT_TO_LREAL(#StepsByMotorTurn) * UINT_TO_LREAL(#StepResolution))/(#MmByMotorTurn*10)));

   #ActualPosition_mm := LREAL_TO_REAL((DINT_TO_LREAL(#Drive_In.P) * TRUNC(#MmByMotorTurn * 100)) / (UINT_TO_LREAL(#StepResolution) * DINT_TO_LREAL(#StepsByMotorTurn)) / 100);
   #IsInAbsolutePosition_1 := "FC10021_TolerenceRelation"(X := #ActualPosition_mm, Y := #AbsolutePosition_1, Tolerance := 1);
   #IsInAbsolutePosition_2 := "FC10021_TolerenceRelation"(X := #ActualPosition_mm, Y := #AbsolutePosition_2, Tolerance := 1);
   #IsInAbsolutePosition_3 := "FC10021_TolerenceRelation"(X := #ActualPosition_mm, Y := #AbsolutePosition_3, Tolerance := 1);
   #IsInAbsolutePosition_4 := "FC10021_TolerenceRelation"(X := #ActualPosition_mm, Y := #AbsolutePosition_4, Tolerance := 1);
   #IsInAbsolutePosition_5 := "FC10021_TolerenceRelation"(X := #ActualPosition_mm, Y := #AbsolutePosition_5, Tolerance := 1);
   #IsInAbsolutePosition_6 := "FC10021_TolerenceRelation"(X := #ActualPosition_mm, Y := #AbsolutePosition_6, Tolerance := 1);
   #IsInAbsolutePosition_7 := "FC10021_TolerenceRelation"(X := #ActualPosition_mm, Y := #AbsolutePosition_7, Tolerance := 1);
   #IsInAbsolutePosition_8 := "FC10021_TolerenceRelation"(X := #ActualPosition_mm, Y := #AbsolutePosition_8, Tolerance := 1);
   #IsInAbsolutePosition_9 := "FC10021_TolerenceRelation"(X := #ActualPosition_mm, Y := #AbsolutePosition_9, Tolerance := 1);
   #IsInAbsolutePosition_10 := "FC10021_TolerenceRelation"(X := #ActualPosition_mm, Y := #AbsolutePosition_10, Tolerance := 1);
END_REGION
END_FUNCTION_BLOCK
